// TIA Portal V20 export
VAR_GLOBAL   // PLC tag table "Marcas programa"
   Tag_1 AT %MB0 : Byte;
   Oihane2 AT %MB53 : Byte;
END_VAR
